FUNCTION LEFTBigString : BOOL

	VAR_INPUT
	pInputString: POINTER TO BYTE;
	SizeOfInputString: UINT;
	SizeToCopy: UINT;
	pOutputString: POINTER TO BYTE;
	SizeOfOutputString: UINT;
END_VAR

VAR
	i: INT;
	pOutputStringNull: POINTER TO BYTE;
END_VAR

(* Make sure output string is big enough to hold the characters *)
IF SizeOfOutputString < SizeToCopy THEN
	RETURN;
END_IF

(* Copy bytes from input string to output string *)
MEMCPY(pOutputString, pInputString, SizeToCopy);

(* Append null character to end of output string *)
pOutputStringNull := (pOutputString + UINT_TO_DINT(SizeToCopy));
pOutputStringNull^ := 0;
LEFTBigString := TRUE;

END_FUNCTION

(* stored: Version 1.1.0.1, ProductVersion 3.1.4024.9
   POU LEFTBigString: Id {456ff1e8-0d9b-43ac-84b1-5e799c58b8bf}, SpecialFunc None *)
